{attribute 'no_check'}
FUNCTION_BLOCK NciChannel_wEvents EXTENDS NciChannel
VAR_INPUT

                        								      
	Event													:	NciEventHandling;
                        	
END_VAR                 	
VAR_OUTPUT              	

END_VAR
VAR
END_VAR

	(* NCI Control											*)
	(********************************************************)

(********************************************************************************)
(* error event ctrl																*)
(********************************************************************************)
	Event(
		Enable			:= ,
		ConfirmTrig		:= NOT Errhdl.flag AND Event.Status.31 OR Admin.ResetAdmin,
		Name			:= ErrHdl.fnc,
		SourceId		:= (* Default *) ,
		rNci			:= THIS^,
		ErrorId			:= TO_UDINT(ErrHdl.Id),
		Status			=> );
		
	(* Reset FB errors by reset flag *)
	(* currently not in use, call _Resetting via state machine to reset Fb errors by setting Execute to FALSE 
	IF Admin.Reset
	THEN
		grp.Execute											:= grp.Execute AND NOT grp.Error;
		itp.Execute											:= itp.Execute AND NOT itp.Error;
		Motion.Execute										:= Motion.Execute AND NOT Motion.Error;
		RPara.Execute										:= RPara.Execute AND NOT RPara.Error;
	END_IF
	*)
	
(********************************************************************************)
(* call super 																	*)
(********************************************************************************)
	SUPER^();
(******************************************************************************)

METHOD reset : Bool
VAR_INPUT
END_VAR

reset 			:= ErrHdl.flag OR SUPER^.reset();
Event.confirm();
END_METHOD

END_FUNCTION_BLOCK

(* stored: Version 1.1.0.1, ProductVersion 3.1.4024.15
   POU NciChannel_wEvents: Id {b92d8dfe-cde0-4af7-8657-957baafaa875}, SpecialFunc None
   Method reset: Id {373d0377-bee3-4867-b2ac-80224d70016d} *)
